Universal Robots PolyScope program: Cobot_soudure_27112023.urp

Program Cobot_soudure_27112023 (installation=Cobot_soudure_27112023 directory=/home/ur/ursim/ursim-5.11.0.108249/programs/TRAVAIL 27112023 createdIn=5.9.4.1031232 lastSavedIn=5.11.0.108249 robotSerialNumber=20195299999)
Calibrated DH parameters: a=[0, -0.6127, -0.57155, 0, 0, 0]; d=[0.1807, 0, 0, 0.17415, 0.11985, 0.11655]; alpha=[1.570796, 0, 0, 1.570796, -1.570796, 0]; deltaTheta=[0, 0, 0, 0, 0, 0]
InitVariablesNode variables(variable(name=Test_Gaz, expression=False), variable(name=Test_Job, expression=False), variable(name=Test_Ordre_Mar, expression=False), variable(name=Valide_Gaz, expression=False), variable(name=fin_soud, expression=1), variable(name=secu_d, expression=0), variable(name=secu_g, expression=0), variable(name=timer_ret_gaz, expression=0))
BeforeStart
  Folder fonctions
    Folder Init [hidden by the author, left out]
    Folder Diverses [hidden by the author, left out]
    Folder Demande [hidden by the author, left out]
    Folder Configuration [hidden by the author, left out]
    Folder Execution [hidden by the author, left out]
    Folder Pas_A_Pas [hidden by the author, left out]
    Folder PopUps
      SuppressedNode
        Folder Configuration [hidden by the author, left out]
      Script file /home/ur/ursim/ursim-5.11.0.108249/programs/SCRIPT/Scripts_soudure/PopUps/Pops_up_PAsAPas.script
        | def pop_up_reg_d():
        |     close_popup()
        |     popup3 = "popup PAS_A_PAS : Table droite programmée"#"popup La table droite est programmée. Appuyer sur le bouton gauche ou droite pour commencer le reglage d'une pièce sur la table associée. La gestion des modes programmation, éxécution et reglage se fait à l'aide des commutateurs superieurs."
        |     socket_open("127.0.0.1",29999,"internal") # open internal socket
        |     socket_send_line(popup3,"internal")     #Affichage message
        |     socket_send_byte(10,"internal")
        | end
        | 
        | def pop_up_reg_g():
        |     close_popup()
        |     popup3 = "popup PAS_A_PAS : Table gauche programmée"#"popup La table gauche est programmée. Appuyer sur le bouton gauche ou droite pour commencer mode pas a pas et le reglage d'une pièce sur la table associée. La gestion des modes programmation, éxécution et reglage se fait à l'aide des commutateurs superieurs."
        |     socket_open("127.0.0.1",29999,"internal") # open internal socket
        |     socket_send_line(popup3,"internal")     #Affichage message
        |     socket_send_byte(10,"internal")
        | end
        | 
        | def pop_up_reg_gd():
        |     close_popup()
        |     popup3 = "popup PAS_A_PAS : Les deux tables sont programmées"#"popup Les deux tables sont programmées. Appuyer sur le bouton gauche ou droite pour commencer le reglage d'une pièce sur la table associée ou passez en mode éxécution à l'aide du commutateur superieur gauche pour effectuer un ou plusieurs cycle(s) de soudure(s)."
        |     socket_open("127.0.0.1",29999,"internal") # open internal socket
        |     socket_send_line(popup3,"internal")     #Affichage message
        |     socket_send_byte(10,"internal")
        | end
        | 
        | def pop_up_reg():
        |     close_popup()
        |     popup3 = "popup PAS_A_PAS : Aucune table n'est programmée"#"popup Appuyer sur le bouton gauche ou droite pour commencer le reglage d'une pièce sur la table associée. La gestion des modes configuration, éxécution et reglage se fait à l'aide des commutateurs superieurs."
        |     socket_open("127.0.0.1",29999,"internal") # open internal socket
        |     socket_send_line(popup3,"internal")     #Affichage message
        |     socket_send_byte(10,"internal")
        | end
        | 
        | def fun_PopUp_PaP(index,type,numPopUP):
        |     index = index +1
        |     char_numeroDeSoudure = to_str(index)
        | 
        |     local resultat = False
        |     local resultat2  = 0
        | 
        |     if (type == 1):
        | 		char_soudure = "point"					#si type = 1, la demande sera sur une soudure point
        | 	elif ((type == 2) or (type ==5)):
        | 		char_soudure = "lineaire"				#si type = 2, la demande sera sur une soudure linéaire
        | 	elif (type == 3):
        | 		char_soudure = "arc de cercle"			#si type = 3, la demande sera sur une soudure arc de cercle
        | 	elif (type == 4):
        | 		char_soudure = "cercle"					#si type = 4, la demande sera sur une soudure cercle
        |     elif (type == 6):
        |         char_soudure = "recopie"                #si type = 5, la demande sera sur une recopie de mouvement
        | 	else :
        | 		char_soudure = "erreur de saisie"
        | 	end
        | 
        |     if (numPopUP == 1):
        |         resultat  = request_boolean_from_primary_client("Soudure numero : " + char_numeroDeSoudure + ", de type : "+ char_soudure + ". Voulez vous effectuer la soudure ?(securité desactivée) Appuyer sur non pour passer à la soudure suivante. ")
        |         return resultat
        |     elif (numPopUP ==2 ):
        |         resultat = request_boolean_from_primary_client("Voulez vous modifier la soudure numéro :" + char_numeroDeSoudure + " ? Appuyez sur non pour continuer")
        |         return resultat
        |     elif (numPopUP ==3 ):
        |         resultat2 = request_integer_from_primary_client("       1-> Point SUIVANT                     Ajouter :    2-> AVANT      3-> APRES")
        |         return resultat2
        |     elif (numPopUP ==4 ):
        |          esultat = request_boolean_from_primary_client("Voulez vous refaire une simulation? Appuyez sur non pour continuer.")
        |         return resultat
        |     end
        | 
        | 
        | end
      Script file /home/ur/ursim/ursim-5.11.0.108249/programs/SCRIPT/Scripts_soudure/PopUps/Pops_up_Execution.script
        | def pop_up_deb_exe_d():
        |     close_popup()
        |     popup3 = "popup Table droite, éxecution... Veillez à bien fermer la porte."
        |     socket_open("127.0.0.1",29999,"internal") # open internal socket
        |     socket_send_line(popup3,"internal")     #Affichage message
        |     socket_send_byte(10,"internal")
        | end
        | 
        | def pop_up_deb_exe_g():
        |     close_popup()
        |     popup3 = "popup Table gauche, éxecution... Veillez à bien fermer la porte."
        |     socket_open("127.0.0.1",29999,"internal") # open internal socket
        |     socket_send_line(popup3,"internal")     #Affichage message
        |     socket_send_byte(10,"internal")
        | end
        | 
        | def pop_up_exe_d():
        |     close_popup()
        |     popup1 = "popup EXECUTION : Table droite prête à éxécution"#"popup Appuyer sur le bouton droit pour commencer l'éxécution de la pièce configurée. La gestion des modes configuration et éxécution se fait à l'aide du commutateur réglage."
        |     socket_open("127.0.0.1",29999,"internal") # open internal socket
        |     socket_send_line(popup1,"internal")     #Affichage message
        |     socket_send_byte(10,"internal")
        | end
        | 
        | def pop_up_exe_g():
        |     close_popup()
        |     popup1 = "popup EXECUTION : Table gauche prête à éxécution"#"popup Appuyer sur le bouton gauche pour commencer l'éxécution de la pièce configurée. La gestion des modes configuration et éxécution se fait à l'aide du commutateur réglage."
        |     socket_open("127.0.0.1",29999,"internal") # open internal socket
        |     socket_send_line(popup1,"internal")     #Affichage message
        |     socket_send_byte(10,"internal")
        | end
        | 
        | def pop_up_fermer_porte():
        |     close_popup()
        |     popup3 = "popup Fermer la porte pour éxecution."
        |     socket_open("127.0.0.1",29999,"internal") # open internal socket
        |     socket_send_line(popup3,"internal")     #Affichage message
        |     socket_send_byte(10,"internal")
        | end
        | 
        | def pop_up_exe():
        |     close_popup()
        |     popup1 ="popup EXECUTION : Les deux tables sont prêtes à l'éxécution" #"popup Appuyer sur le bouton gauche ou droit pour commencer l'éxécution de la pièce sur la table associée. La gestion des modes configuration et éxécution se fait à l'aide du commutateur réglage."
        |     socket_open("127.0.0.1",29999,"internal") # open internal socket
        |     socket_send_line(popup1,"internal")     #Affichage message
        |     socket_send_byte(10,"internal")
        | end
      Script file /home/ur/ursim/ursim-5.11.0.108249/programs/SCRIPT/Scripts_soudure/PopUps/Pops_up_Configuration.script
        | def pop_up_config():
        |     close_popup()
        |     popup3 = "popup CONFIGURATION : Aucune table de configurée."
        |     socket_open("127.0.0.1",29999,"internal") # open internal socket
        |     socket_send_line(popup3,"internal")     #Affichage message
        |     socket_send_byte(10,"internal")
        | end
        | 
        | def pop_up_config_d():
        |     close_popup()
        |     popup3 = "popup CONFIGURATION : Table droite configurée."
        |     socket_open("127.0.0.1",29999,"internal") # open internal socket
        |     socket_send_line(popup3,"internal")     #Affichage message
        |     socket_send_byte(10,"internal")
        | end
        | 
        | def pop_up_config_g_et_d():
        |     close_popup()
        |     popup3 = "popup CONFIGURATION : Les deux tables sont configurées."
        |     socket_open("127.0.0.1",29999,"internal") # open internal socket
        |     socket_send_line(popup3,"internal")     #Affichage message
        |     socket_send_byte(10,"internal")
        | end
        | 
        | def pop_up_config_g():
        |     close_popup()
        |     popup3 = "popup CONFIGURATION : Table droite configurée."
        |     socket_open("127.0.0.1",29999,"internal") # open internal socket
        |     socket_send_line(popup3,"internal")     #Affichage message
        |     socket_send_byte(10,"internal")
        | end
      SuppressedNode
        Folder Execution [hidden by the author, left out]
      SuppressedNode
        Folder Pas_A_Pas [hidden by the author, left out]
    Folder Mouvements soudures [hidden by the author, left out]
Robot Program (runOnlyOnce=true)
  SuppressedNode
    Folder Initialisation
      Loop Counting (count=1) loopVariable(name=Boucle_10)
        Script: fun_adresse_bp()
  Script file /home/ur/ursim/ursim-5.11.0.108249/programs/SCRIPT/Scripts_soudure/general.script
    | while (True):
    |   # 68 "Programme de robot"
    |   global safe_mode=0
    | 
    |   set_configurable_digital_out(0, False)
    | 
    |   set_configurable_digital_out(1, False)
    | 
    |   while (get_configurable_digital_in(4) ==   True    or  get_configurable_digital_in(5) ==   True  ):
    | 
    |     sync()
    |     # 94 "'clingottement pour signifier qu'il y  un defaut sur un des carters '"
    |     set_standard_digital_out(4, False)
    |     set_configurable_digital_out(6, False)
    |     sleep(0.5)
    |     set_standard_digital_out(4, True)
    |     set_configurable_digital_out(6, True)
    |     sleep(0.5)
    |     sync()
    |   end
    | 
    |   set_configurable_digital_out(6, False)
    |   set_standard_digital_out(4, False)
    |   sleep(2.0)
    |   #movel(pose_add(get_target_tcp_pose(), pose_sub(PointPassage_12_to_p, PointPassage_12_from_p)), a=0.01, v=2.0E-4)
    |   global angle_base= get_actual_joint_positions ()
    |   if (angle_base[0]  <= 0.7):
    |     if (angle_base[0] >= 1.6):
    |       # 116 "Départ"        A CHANGER PAR UNE POSTION ENREGISTREE
    |       movej([0.7376820445060732, 1.3357652919721463, -2.8533326461405863, -0.44459326684985356, 1.9245067834854124, 4.003490924835204], a=1.3962634015954636, v=1.0471975511965976)
    |     else:
    |       if (angle_base[0]>1.6):
    |         movej(Point_init_D, a=1.3962634015954636, v=1.7453292519943295)
    |         movej(Point_avt_initD, a=1.3962634015954636, v=1.7453292519943295)
    |       else:
    |         if (angle_base[0]<0.7):
    |           movej(Point_init_G, a=1.3962634015954636, v=1.7453292519943295)
    |         end
    |       end
    |     end
    |   else:
    |     # 124 "SinonSi angle_base[0]>1.6"
    |     if (angle_base[0]>1.6):
    | 
    |       movej(Point_init_D, a=1.3962634015954636, v=1.7453292519943295)
    |       movej(Point_avt_initD, a=1.3962634015954636, v=1.7453292519943295)
    |     else:
    |       if (angle_base[0]<0.7):
    |         movej(Point_init_G, a=1.3962634015954636, v=1.7453292519943295)
    |       end
    |     end
    |   end
    |   # 131 "Départ"             A CHANGER PAR UNE POSTION ENREGISTREE
    |   movej([0.7376820445060732, 1.3357652919721463, -2.8533326461405863, -0.44459326684985356, 1.9245067834854124, 4.003490924835204], a=1.3962634015954636, v=1.0471975511965976)
    |   global angle_base= get_actual_joint_positions ()
    |   # 'mode config'
    |   if (get_configurable_digital_in(7)  ==   False    and  get_standard_digital_in(7)  ==   False  ):
    |     if ((config_g  ==  1)   and   (config_d  ==  1)):
    |       pop_up_config_g_et_d()
    |     else:
    |       if ((config_g  == 1)):
    |         pop_up_config_g()
    |       else:
    |         if (config_d  ==  1):
    |           pop_up_config_d()
    |         else:
    |           if ((config_g  ==  0)  and  (config_d  ==  0)):
    |             pop_up_config()
    |           end
    |         end
    |       end
    |     end
    |     global boucle=1
    |     while ((get_configurable_digital_in(7)  ==   False  )  and  (boucle  ==  1)   and  (get_standard_digital_in(7) ==   False  )):
    |       thread Thread_while_145():
    |         while (True):
    |           set_standard_digital_out(5, True)
    |           set_standard_digital_out(6, False)
    |           sleep(0.5)
    |           set_standard_digital_out(5, False)
    |           set_standard_digital_out(6, True)
    |           sleep(0.5)
    |           sync()
    |         end
    |       end
    |       if (get_standard_digital_in(3) ==   False    and  get_standard_digital_in(2) ==   False    and  get_configurable_digital_in(7)  ==    False    and  get_standard_digital_in(7) ==   False  ):
    |         global thread_handler_145=run Thread_while_145()
    |         while (get_standard_digital_in(3) ==   False    and  get_standard_digital_in(2) ==   False    and  get_configurable_digital_in(7)  ==    False    and  get_standard_digital_in(7) ==   False  ):
    |           sync()
    |         end
    |         kill thread_handler_145
    |       end
    |       if (get_standard_digital_in(2)  ==   True  ):
    |         set_standard_digital_out(5, True)
    |         set_standard_digital_out(6, False)
    |         movej(Point_init_G, a=1.3962634015954636, v=1.0471975511965976, r=0.006)
    |         movej(Point_Attente_G, a=1.3962634015954636, v=1.0471975511965976, r=0.006)
    |         movej(Point_config_g, a=0.6981317007977318, v=0.5235987755982988)
    |         global led_cobot=1
    |         fun_config_g()
    |         global led_cobot=0
    |         fun_valid_config_g()
    |         movej(Point_Attente_G, a=1.3962634015954636, v=1.0471975511965976, r=0.006)
    |         movej(Point_init_G, a=1.3962634015954636, v=1.0471975511965976, r=0.006)
    |         # 170 "Départ"         A CHANGER PAR UNE POSTION ENREGISTREE
    |         movej([0.7376820445060732, 1.3357652919721463, -2.8533326461405863, -0.44459326684985356, 1.9245067834854124, 4.003490924835204], a=1.3962634015954636, v=1.0471975511965976)
    |       end
    | 
    |       if (get_standard_digital_in(3)  ==   True  ):
    |         set_standard_digital_out(6, True)
    |         set_standard_digital_out(5, False)
    |         movej(Point_avt_initD, a=1.3962634015954636, v=1.0471975511965976, r=0.006)
    |         movej(Point_init_D, a=1.3962634015954636, v=1.0471975511965976)
    |         movej(Point_Attente_D, a=1.3962634015954636, v=1.0471975511965976, r=0.006)
    |         movej(Point_config_d, a=0.6981317007977318, v=0.5235987755982988)
    |         global led_cobot=1
    |         fun_config_d()
    |         global led_cobot=0
    |         fun_valid_config_d()
    |         movej(Point_Attente_D, a=1.3962634015954636, v=1.0471975511965976, r=0.006)
    |         movej(Point_init_D, a=1.3962634015954636, v=1.0471975511965976, r=0.006)
    |         movej(Point_avt_initD, a=1.3962634015954636, v=1.0471975511965976, r=0.006)
    |         # 190 "Départ"         A CHANGER PAR UNE POSTION ENREGISTREE
    |         movej([0.7376820445060732, 1.3357652919721463, -2.8533326461405863, -0.44459326684985356, 1.9245067834854124, 4.003490924835204], a=1.3962634015954636, v=1.0471975511965976)
    |       end
    |     end
    |   end
    |   # '"Reglage"'
    | 
    |   if (get_configurable_digital_in(7)  ==   False    and  get_standard_digital_in(7)  ==   True  ):
    |     if ((config_g  ==  1)   and   (config_d  ==  1)):
    |       pop_up_reg_gd()
    |       global boucle=1
    |     else:
    |       if (config_g  ==  1):
    |         pop_up_reg_gd()
    |         global boucle=1
    |       else:
    |         if (config_d  ==  1):
    |           pop_up_reg_d()
    |           global boucle=1
    |         else:
    |           close_popup()
    |           while (get_standard_digital_in(7)  ==   True  ):
    |             popup("Aucune configuration n'est actuellement detectée.", "Erreur", False, True, blocking=True)
    |           end
    |         end
    |       end
    |     end
    |     global boucle=1
    |     while ((get_configurable_digital_in(7)  ==   False  )  and  (boucle  ==  1)   and  (get_standard_digital_in(7) ==   True  )):
    |       thread Thread_while_208():
    |         while (True):
    |           if (config_g  ==  1):
    |             set_standard_digital_out(5, True)
    |           end
    |           if (config_d  ==  1):
    |             set_standard_digital_out(6, True)
    |           end
    |           sleep(0.5)
    |           set_standard_digital_out(5, False)
    |           set_standard_digital_out(6, False)
    |           sleep(0.5)
    |         end
    |       end
    |       if (get_standard_digital_in(3) ==   False    and  get_standard_digital_in(2) ==   False    and  get_configurable_digital_in(7)  ==    False    and  get_standard_digital_in(7)  ==   True  ):
    |         global thread_handler_208=run Thread_while_208()
    |         while (get_standard_digital_in(3) ==   False    and  get_standard_digital_in(2) ==   False    and  get_configurable_digital_in(7)  ==    False    and  get_standard_digital_in(7)  ==   True  ):
    |           sync()
    |         end
    |         kill thread_handler_208
    |       end
    |       if (get_standard_digital_in(2)  ==   True  ):
    |         global safe_mode=1
    |         set_standard_digital_out(5, True)
    |         set_standard_digital_out(6, False)
    |         movej(Point_init_G, a=1.3962634015954636, v=1.0471975511965976, r=0.006)
    |         movej(Point_Attente_G, a=1.3962634015954636, v=1.0471975511965976, r=0.006)
    |         movej(pose_inter_g, a=0.6981317007977318, v=0.5235987755982988)
    |         global led_cobot=1
    |         fun_Pas_A_Pas_g()
    |         global led_cobot=0
    |         global safe_mode=0
    |         global boucle=0
    |       end
    |       if (get_standard_digital_in(3)  ==   True  ):
    |         global safe_mode=1
    |         set_standard_digital_out(6, True)
    |         set_standard_digital_out(5, False)
    |         movej(Point_avt_initD, a=1.3962634015954636, v=1.0471975511965976, r=0.006)
    |         movej(Point_init_D, a=1.3962634015954636, v=1.0471975511965976, r=0.006)
    |         movej(pose_inter_d, a=0.6981317007977318, v=0.5235987755982988)
    |         global led_cobot=1
    |         fun_Pas_A_Pas_d()
    |         global led_cobot=0
    |         global safe_mode=0
    |         global boucle=0
    |       end
    |     end
    |   end
    |   # 'mode execution'
    |   if (get_configurable_digital_in(7)  ==   True  ):
    |     if ((config_g  ==  1)   and   (config_d  ==  1)):
    |       pop_up_exe()
    |       global boucle=1
    |     else:
    |       if (config_g  ==  1):
    |         pop_up_exe_g()
    |         global boucle=1
    |       else:
    |         if (config_d  ==  1):
    |           pop_up_exe_d()
    |           global boucle=1
    |         else:
    |           close_popup()
    |           while (get_configurable_digital_in(7)  ==   True  ):
    |             popup("Aucune programmation n'est actuellement detectée, veillez à programmer une pièce avant de vouloir l'éxécuter.", "Erreur", False, True, blocking=True)
    |           end
    |         end
    |       end
    |     end
    |     while (( get_configurable_digital_in(7)  ==   True  )   and  (boucle  ==  1)):
    |       thread Thread_while_259():
    |         while (True):
    |           if (config_g  ==  1):
    |             set_standard_digital_out(5, True)
    |           end
    |           if (config_d  ==  1):
    |             set_standard_digital_out(6, True)
    |           end
    |           sleep(0.5)
    |           set_standard_digital_out(5, False)
    |           set_standard_digital_out(6, False)
    |           sleep(0.5)
    |         end
    |       end
    |       if (get_standard_digital_in(3) ==   False    and  get_standard_digital_in(2) ==   False    and  get_configurable_digital_in(7) ==   True  ):
    |         global thread_handler_259=run Thread_while_259()
    |         while (get_standard_digital_in(3) ==   False    and  get_standard_digital_in(2) ==   False    and  get_configurable_digital_in(7) ==   True  ):
    |           sync()
    |         end
    |         kill thread_handler_259
    |       end
    |       if ((get_standard_digital_in(2)  ==   True  )  and  (config_g  ==   True  )):
    |         global boucle_g=1
    |         while (boucle_g  ==  1):
    |           set_configurable_digital_out(0, True)
    |           set_standard_digital_out(5, True)
    |           set_standard_digital_out(6, False)
    |           sleep(0.25)
    |           set_standard_digital_out(5, False)
    |           sleep(0.25)
    |           if (get_configurable_digital_in(4)  ==    False  ):
    |             set_standard_digital_out(5, True)
    |             if (get_configurable_digital_in(4)  ==    False  ):
    |               close_popup()
    |               while (get_configurable_digital_in(4) == False):
    |                 sync()
    |               end
    |             end
    |           end
    |           if (get_configurable_digital_in(4)  ==    True  ):
    |             global secu_g=1
    |             set_standard_digital_out(5, True)
    |             movej(Point_init_G, a=1.3962634015954636, v=1.0471975511965976, r=0.006)
    |             fun_execution_g()
    |             movej(Point_Attente_G, a=1.3962634015954636, v=1.0471975511965976, r=0.006)
    |             movej(Point_init_G, a=1.3962634015954636, v=1.0471975511965976, r=0.006)
    |             # 294 "Départ"         A CHANGER PAR UNE POSTION ENREGISTREE
    |             movej([0.7376820445060732, 1.3357652919721463, -2.8533326461405863, -0.44459326684985356, 1.9245067834854124, 4.003490924835204], a=1.3962634015954636, v=1.0471975511965976)
    |             set_configurable_digital_out(0, False)
    |             global secu_g=0
    |             global boucle_g=0
    |           end
    |         end
    |         global boucle=0
    |       else:
    |         if ((get_standard_digital_in(2)  ==   True  )  and  (config_g  ==   False  )):
    |           close_popup()
    |           popup("Aucune programmation n'est actuellement detectée sur la table gauche, veillez à programmer une pièce avant de vouloir l'éxécuter.", "Erreur", False, True, blocking=True)
    |           global boucle=0
    |         end
    |       end
    |       if ((get_standard_digital_in(3)  ==   True  )  and  (config_d  ==   True  )):
    |         global boucle_d=1
    |         pop_up_deb_exe_d()
    |         while (boucle_d  ==  1):
    |           set_configurable_digital_out(1, True)
    |           set_standard_digital_out(5, False)
    |           set_standard_digital_out(6, True)
    |           sleep(0.25)
    |           set_standard_digital_out(6, False)
    |           sleep(0.25)
    |           if (get_configurable_digital_in(5)  ==    False  ):
    |             set_standard_digital_out(6, True)
    |             sleep(6.0)
    |             if (get_configurable_digital_in(5)  ==    False  ):
    |               close_popup()
    |               while (get_configurable_digital_in(5) == False):
    |                 sync()
    |               end
    |             end
    |           end
    |           if (get_configurable_digital_in(5)  ==    True  ):
    |             global secu_d=1
    |             set_standard_digital_out(6, True)
    |             movej(Point_avt_initD, a=1.3962634015954636, v=1.0471975511965976)
    |             fun_execution_d()
    |             set_configurable_digital_out(1, False)
    |             global secu_d=0
    |             global boucle_d=0
    |           end
    |         end
    |         global boucle=0
    |       else:
    |         if ((get_standard_digital_in(3)  ==   True  )  and  (config_d  ==   False  )):
    |           close_popup()
    |           popup("Aucune programmation n'est actuellement detectée sur la table droite, veillez à programmer une pièce avant de vouloir l'éxécuter.", "Erreur", False, True, blocking=True)
    |           global boucle=0
    |         end
    |       end
    |     end
    |   end
    | end
    | end
  SuppressedNode
    MoveJ speed 60 deg/s, acceleration 80 deg/s^2 (useActiveTCP=true) feature=Base
      SafeHome (positionOptionType=SPEED_AND_ACCELERATION speed=1.047198 acceleration=1.396263 nextMotionTime=2)
      Waypoint Waypoint (Variable): motionParameters(jointSpeed=0.523599 jointAcceleration=0.698132 cartesianSpeed=0.25 cartesianAcceleration=1.2); variable(featureName=Point_init_G)
      Waypoint Waypoint (Variable): motionParameters(jointSpeed=0.523599 jointAcceleration=0.698132 cartesianSpeed=0.25 cartesianAcceleration=1.2); variable(featureName=Point_Attente_G)
      Waypoint Waypoint (Variable): motionParameters(jointSpeed=0.523599 jointAcceleration=0.698132 cartesianSpeed=0.25 cartesianAcceleration=1.2); variable(featureName=Point_config_g)
      Waypoint Waypoint (Variable): motionParameters(jointSpeed=0.523599 jointAcceleration=0.698132 cartesianSpeed=0.25 cartesianAcceleration=1.2); variable(featureName=Point_Attente_G)
      Waypoint Waypoint (Variable): motionParameters(jointSpeed=0.523599 jointAcceleration=0.698132 cartesianSpeed=0.25 cartesianAcceleration=1.2); variable(featureName=Point_init_G)
      SafeHome (positionOptionType=SPEED_AND_ACCELERATION speed=1.047198 acceleration=1.396263 nextMotionTime=2)
      Waypoint Waypoint (Variable): motionParameters(jointSpeed=0.785398 jointAcceleration=1.047198 cartesianSpeed=0.25 cartesianAcceleration=1.2); variable(featureName=Point_avt_initD)
      Waypoint Waypoint (Variable): motionParameters(jointSpeed=0.523599 jointAcceleration=0.698132 cartesianSpeed=0.25 cartesianAcceleration=1.2); variable(featureName=Point_init_D)
      Waypoint Waypoint (Variable): motionParameters(jointSpeed=0.523599 jointAcceleration=0.698132 cartesianSpeed=0.25 cartesianAcceleration=1.2); variable(featureName=Point_Attente_D)
      Waypoint Waypoint (Variable): motionParameters(jointSpeed=0.523599 jointAcceleration=0.698132 cartesianSpeed=0.25 cartesianAcceleration=1.2); variable(featureName=Point_config_d)
      Waypoint Waypoint (Variable): motionParameters(jointSpeed=0.523599 jointAcceleration=0.698132 cartesianSpeed=0.25 cartesianAcceleration=1.2); variable(featureName=Point_Attente_D)
      Waypoint Waypoint (Variable): motionParameters(jointSpeed=0.523599 jointAcceleration=0.698132 cartesianSpeed=0.25 cartesianAcceleration=1.2); variable(featureName=Point_init_D)
      SafeHome (positionOptionType=SPEED_AND_ACCELERATION speed=1.047198 acceleration=1.396263 nextMotionTime=2)
  SuppressedNode
    safe_mode := 0
  SuppressedNode
    Folder Deplacement vers position initial
      SuppressedNode
        Popup Message (haltProgram=false message=debut deplacement vers position initiale inputType=Text)
      Set DigitalOutput pin=Cmd_Carter_Bit1; digitalValue=0
      Set DigitalOutput pin=Cmd_Carter_Bit2; digitalValue=0
      Loop While (checkContinuously=false) expression=SecuGaucheOk≟ True  or SecuDroiteOk≟ True
        Script: sync()
        'clingottement pour signifier qu'il y  un defaut sur un des carters '
        Set DigitalOutput pin=Dcy_Voyant; digitalValue=0
        Set DigitalOutput pin=Led_Arret; digitalValue=0
        Wait Sleep waitTime=0.5
        Set DigitalOutput pin=Dcy_Voyant; digitalValue=1
        Set DigitalOutput pin=Led_Arret; digitalValue=1
        Wait Sleep waitTime=0.5
      Set DigitalOutput pin=Led_Arret; digitalValue=0
      Set DigitalOutput pin=Dcy_Voyant; digitalValue=0
      Wait Sleep waitTime=2
      'etre sur de l'ouverture complete du carter '
      MoveL speed 0.2 mm/s, acceleration 10 mm/s^2 (useActiveTCP=true) feature=Base
        Waypoint PointPassage_12 (Relative): relativeFromPosition TCP in base x=100.468 y=319.613 z=576.47 mm, rx=-0.0214 ry=-0.0122 rz=1.5415 rad; joints [-139.419, 75.739, -163.156, -3.26, 89.083, -42.172] deg; TCP offset x=-8.331 y=2.512 z=301.573 mm, rx=0 ry=0 rz=0 rad; TCP in base x=100.463 y=319.639 z=576.462 mm, rx=-0.0214 ry=-0.0122 rz=1.5416 rad; joints [-139.419, 75.741, -163.155, -3.263, 89.08, -42.17] deg
        'Pos_cobot a etait affectuer a la position init (l3)'
        'Pos_cobot[2] correspond a la valeur Z de la postion init (l4)'
      SuppressedNode
        MoveJ speed 60 deg/s, acceleration 80 deg/s^2 (useActiveTCP=true) feature=Base
          SuppressedNode
            Waypoint Position_init: motionParameters(jointSpeed=1.047198 jointAcceleration=1.396263 cartesianSpeed=0.25 cartesianAcceleration=1.2); TCP in base x=96.613 y=317.698 z=575.432 mm, rx=-0.0254 ry=-0.0254 rz=1.5393 rad; joints [-139.566, 75.575, -163.284, -3.665, 88.92, -42.143] deg; TCP offset x=-6.782 y=1.742 z=298.685 mm, rx=0 ry=0 rz=0 rad
          SuppressedNode
            Waypoint Waypoint (Variable): variable(featureName=Point_init)
          'Apres avoir eu la position du robot et tester la valeur de Z pour faire un mouvement verticale on envoi le robot en position init'
      angle_base := get_actual_joint_positions()
      If angle_base[0] ≤0.7
        If angle_base[0]≥1.6
          SafeHome (positionOptionType=SPEED_AND_ACCELERATION speed=1.047198 acceleration=1.396263 nextMotionTime=2)
        ElseIf angle_base[0]>1.6
          MoveJ speed 100 deg/s, acceleration 80 deg/s^2 (useActiveTCP=true) feature=Base
            Waypoint Waypoint (Variable): variable(featureName=Point_init_D)
            Waypoint Waypoint (Variable): variable(featureName=Point_avt_initD)
        ElseIf angle_base[0]<0.7
          MoveJ speed 100 deg/s, acceleration 80 deg/s^2 (useActiveTCP=true) feature=Base
            Waypoint Waypoint (Variable): variable(featureName=Point_init_G)
      ElseIf angle_base[0]>1.6
        MoveJ speed 100 deg/s, acceleration 80 deg/s^2 (useActiveTCP=true) feature=Base
          Waypoint Waypoint (Variable): variable(featureName=Point_init_D)
          Waypoint Waypoint (Variable): variable(featureName=Point_avt_initD)
      ElseIf angle_base[0]<0.7
        MoveJ speed 100 deg/s, acceleration 80 deg/s^2 (useActiveTCP=true) feature=Base
          Waypoint Waypoint (Variable): variable(featureName=Point_init_G)
      SafeHome (positionOptionType=SPEED_AND_ACCELERATION speed=1.047198 acceleration=1.396263 nextMotionTime=2)
      angle_base := get_actual_joint_positions()
  SuppressedNode
    'mode config'
  SuppressedNode
    If Mode_manu ≟ False  and config_reglage ≟ False
      If (config_g ≟ 1)  and  (config_d ≟ 1)
        Script: pop_up_config_g_et_d()
      ElseIf (config_g ≟1)
        Script: pop_up_config_g()
      ElseIf config_d ≟ 1
        Script: pop_up_config_d()
      ElseIf (config_g ≟ 0) and (config_d ≟ 0)
        Script: pop_up_config()
      boucle := 1
      Loop While (checkContinuously=false) expression=(Mode_manu ≟ False ) and (boucle ≟ 1)  and (config_reglage≟ False )
        Loop While (checkContinuously=true) expression=Pret_Table_Droi≟ False  and Pret_Table_Gauc≟ False  and Mode_manu ≟  False  and config_reglage≟ False
          Set DigitalOutput pin=Voyant_Table_Ga; digitalValue=1
          Set DigitalOutput pin=Voyant_Table_Dr; digitalValue=0
          Wait Sleep waitTime=0.5
          Set DigitalOutput pin=Voyant_Table_Ga; digitalValue=0
          Set DigitalOutput pin=Voyant_Table_Dr; digitalValue=1
          Wait Sleep waitTime=0.5
          Script: sync()
        If Pret_Table_Gauc ≟ True
          Set DigitalOutput pin=Voyant_Table_Ga; digitalValue=1
          Set DigitalOutput pin=Voyant_Table_Dr; digitalValue=0
          'plus de demande du nombre de point a saisir'
          MoveJ speed 60 deg/s, acceleration 80 deg/s^2 (useActiveTCP=true) feature=Base
            Waypoint Waypoint (Variable): motionParameters(blendRadius=0.006); variable(featureName=Point_init_G)
            Waypoint Waypoint (Variable): motionParameters(blendRadius=0.006); variable(featureName=Point_Attente_G)
            Waypoint Waypoint (Variable): motionParameters(jointSpeed=0.523599 jointAcceleration=0.698132 cartesianSpeed=0.25 cartesianAcceleration=1.2); variable(featureName=Point_config_g)
            led_cobot := 1
            Script: fun_config_g()
            led_cobot := 0
            Script: fun_valid_config_g()
            MoveJ speed 60 deg/s, acceleration 80 deg/s^2 (useActiveTCP=true) feature=Base
              SuppressedNode
                Waypoint anti_poq_g: motionParameters(jointSpeed=0.523599 jointAcceleration=0.698132 cartesianSpeed=0.25 cartesianAcceleration=1.2 blendRadius=0.07); TCP in base x=433.126 y=153.22 z=577.202 mm, rx=0.0572 ry=-0.0147 rz=1.5652 rad; joints [-179.123, 70.738, -150.145, -9.057, 92.825, -1.059] deg; TCP offset x=-8.331 y=2.512 z=301.573 mm, rx=0 ry=0 rz=0 rad
              Waypoint Waypoint (Variable): motionParameters(blendRadius=0.006); variable(featureName=Point_Attente_G)
              Waypoint Waypoint (Variable): motionParameters(blendRadius=0.006); variable(featureName=Point_init_G)
              SuppressedNode
                Waypoint Waypoint (Variable): motionParameters(jointSpeed=0.523599 jointAcceleration=0.698132 cartesianSpeed=0.25 cartesianAcceleration=1.2); variable(featureName=Point_init)
              SafeHome (positionOptionType=SPEED_AND_ACCELERATION speed=1.047198 acceleration=1.396263 nextMotionTime=2)
        If Pret_Table_Droi ≟ True
          Set DigitalOutput pin=Voyant_Table_Dr; digitalValue=1
          Set DigitalOutput pin=Voyant_Table_Ga; digitalValue=0
          MoveJ speed 60 deg/s, acceleration 80 deg/s^2 (useActiveTCP=true) feature=Base
            Waypoint Waypoint (Variable): motionParameters(blendRadius=0.006); variable(featureName=Point_avt_initD)
            Waypoint Waypoint (Variable): variable(featureName=Point_init_D)
            Waypoint Waypoint (Variable): motionParameters(blendRadius=0.006); variable(featureName=Point_Attente_D)
            Waypoint Waypoint (Variable): motionParameters(jointSpeed=0.523599 jointAcceleration=0.698132 cartesianSpeed=0.25 cartesianAcceleration=1.2); variable(featureName=Point_config_d)
          led_cobot := 1
          Script: fun_config_d()
          led_cobot := 0
          Script: fun_valid_config_d()
          MoveJ speed 60 deg/s, acceleration 80 deg/s^2 (useActiveTCP=true) feature=Base
            SuppressedNode
              Waypoint anti_poq_1_d: motionParameters(jointSpeed=0.523599 jointAcceleration=0.698132 cartesianSpeed=0.25 cartesianAcceleration=1.2 blendRadius=0); TCP in base x=-432.081 y=47.828 z=581.386 mm, rx=0.0024 ry=-0.0004 rz=1.5709 rad; joints [-31.202, 71.743, -153.151, -8.683, 90.121, -148.72] deg
            SuppressedNode
              Waypoint anti_poq_2_d: motionParameters(jointSpeed=1.047198 jointAcceleration=1.396263 cartesianSpeed=0.25 cartesianAcceleration=1.2 blendRadius=0.07); TCP in base x=-292.604 y=310.313 z=583.956 mm, rx=-0.0324 ry=-0.0877 rz=3.0963 rad; joints [-72.124, 71.739, -151.869, -12.519, 87.987, -20.279] deg; TCP offset x=-8.331 y=2.512 z=301.573 mm, rx=0 ry=0 rz=0 rad
            SuppressedNode
              Waypoint Waypoint (Variable): motionParameters(jointSpeed=0.785398 jointAcceleration=1.047198 cartesianSpeed=0.25 cartesianAcceleration=1.2); variable(featureName=Point_init)
            Waypoint Waypoint (Variable): motionParameters(blendRadius=0.006); variable(featureName=Point_Attente_D)
            Waypoint Waypoint (Variable): motionParameters(blendRadius=0.006); variable(featureName=Point_init_D)
            Waypoint Waypoint (Variable): motionParameters(blendRadius=0.006); variable(featureName=Point_avt_initD)
            SafeHome (positionOptionType=SPEED_AND_ACCELERATION speed=1.047198 acceleration=1.396263 nextMotionTime=2)
  SuppressedNode
    '"Reg"'
  SuppressedNode
    If Mode_manu ≟ False  and config_reglage ≟ True
      If (config_g ≟ 1)  and  (config_d ≟ 1)
        Script: pop_up_reg_gd()
        boucle := 1
      ElseIf config_g ≟ 1
        Script: pop_up_reg_gd()
        boucle := 1
      ElseIf config_d ≟ 1
        Script: pop_up_reg_d()
        boucle := 1
      Else 
        Script: close_popup()
        Loop While (checkContinuously=false) expression=config_reglage ≟ True
          Popup Error (haltProgram=false message=Aucune configuration n'est actuellement detectée. inputType=Text)
      boucle := 1
      Loop While (checkContinuously=false) expression=(Mode_manu ≟ False ) and (boucle ≟ 1)  and (config_reglage≟ True )
        Loop While (checkContinuously=true) expression=Pret_Table_Droi≟ False  and Pret_Table_Gauc≟ False  and Mode_manu ≟  False  and config_reglage ≟ True
          If config_g ≟ 1
            Set DigitalOutput pin=Voyant_Table_Ga; digitalValue=1
          If config_d ≟ 1
            Set DigitalOutput pin=Voyant_Table_Dr; digitalValue=1
          Wait Sleep waitTime=0.5
          Set DigitalOutput pin=Voyant_Table_Ga; digitalValue=0
          Set DigitalOutput pin=Voyant_Table_Dr; digitalValue=0
          Wait Sleep waitTime=0.5
        If Pret_Table_Gauc ≟ True
          safe_mode := 1
          Set DigitalOutput pin=Voyant_Table_Ga; digitalValue=1
          Set DigitalOutput pin=Voyant_Table_Dr; digitalValue=0
          MoveJ speed 60 deg/s, acceleration 80 deg/s^2 (useActiveTCP=true) feature=Base
            Waypoint Waypoint (Variable): motionParameters(blendRadius=0.006); variable(featureName=Point_init_G)
            Waypoint Waypoint (Variable): motionParameters(blendRadius=0.006); variable(featureName=Point_Attente_G)
            Waypoint Waypoint (Variable): motionParameters(jointSpeed=0.523599 jointAcceleration=0.698132 cartesianSpeed=0.25 cartesianAcceleration=1.2); variable(featureName=pose_inter_g)
          led_cobot := 1
          Script: fun_Pas_A_Pas_g()
          led_cobot := 0
          safe_mode := 0
          boucle := 0
        If Pret_Table_Droi ≟ True
          safe_mode := 1
          Set DigitalOutput pin=Voyant_Table_Dr; digitalValue=1
          Set DigitalOutput pin=Voyant_Table_Ga; digitalValue=0
          MoveJ speed 60 deg/s, acceleration 80 deg/s^2 (useActiveTCP=true) feature=Base
            Waypoint Waypoint (Variable): motionParameters(blendRadius=0.006); variable(featureName=Point_avt_initD)
            Waypoint Waypoint (Variable): motionParameters(blendRadius=0.006); variable(featureName=Point_init_D)
            Waypoint Waypoint (Variable): motionParameters(jointSpeed=0.523599 jointAcceleration=0.698132 cartesianSpeed=0.25 cartesianAcceleration=1.2); variable(featureName=pose_inter_d)
          led_cobot := 1
          Script: fun_Pas_A_Pas_d()
          led_cobot := 0
          safe_mode := 0
          boucle := 0
  SuppressedNode
    'mode exe'
  SuppressedNode
    If Mode_manu ≟ True
      If (config_g ≟ 1)  and  (config_d ≟ 1)
        Script: pop_up_exe()
        boucle := 1
      ElseIf config_g ≟ 1
        Script: pop_up_exe_g()
        boucle := 1
      ElseIf config_d ≟ 1
        Script: pop_up_exe_d()
        boucle := 1
      Else 
        Script: close_popup()
        Loop While (checkContinuously=false) expression=Mode_manu ≟ True
          Popup Error (haltProgram=false message=Aucune programmation n'est actuellement detectée, veillez à programmer une pièce avant de vouloir l'éxécuter. inputType=Text)
      Loop While (checkContinuously=false) expression=( Mode_manu ≟ True )  and (boucle ≟ 1)
        Loop While (checkContinuously=true) expression=Pret_Table_Droi≟ False  and Pret_Table_Gauc≟ False  and Mode_manu≟ True
          If config_g ≟ 1
            Set DigitalOutput pin=Voyant_Table_Ga; digitalValue=1
          If config_d ≟ 1
            Set DigitalOutput pin=Voyant_Table_Dr; digitalValue=1
          Wait Sleep waitTime=0.5
          Set DigitalOutput pin=Voyant_Table_Ga; digitalValue=0
          Set DigitalOutput pin=Voyant_Table_Dr; digitalValue=0
          Wait Sleep waitTime=0.5
        If (Pret_Table_Gauc ≟ True ) and (config_g ≟ True )
          boucle_g := 1
          SuppressedNode
            Script: pop_up_deb_exe_g()
          Loop While (checkContinuously=false) expression=boucle_g ≟ 1
            Set DigitalOutput pin=Cmd_Carter_Bit1; digitalValue=1
            Set DigitalOutput pin=Voyant_Table_Ga; digitalValue=1
            Set DigitalOutput pin=Voyant_Table_Dr; digitalValue=0
            Wait Sleep waitTime=0.25
            Set DigitalOutput pin=Voyant_Table_Ga; digitalValue=0
            Wait Sleep waitTime=0.25
            If SecuGaucheOk ≟  False
              Set DigitalOutput pin=Voyant_Table_Ga; digitalValue=1
              SuppressedNode
                Wait Sleep waitTime=6
              If SecuGaucheOk ≟  False
                Script: close_popup()
                Wait DigitalInput pin=SecuGaucheOk; digitalValue=1
            If SecuGaucheOk ≟  True
              secu_g := 1
              Set DigitalOutput pin=Voyant_Table_Ga; digitalValue=1
              MoveJ speed 60 deg/s, acceleration 80 deg/s^2 (useActiveTCP=true) feature=Base
                Waypoint Waypoint (Variable): motionParameters(blendRadius=0.006); variable(featureName=Point_init_G)
                SuppressedNode
                  Waypoint Waypoint (Variable): motionParameters(blendRadius=0.006); variable(featureName=Point_Attente_G)
              Script: fun_execution_g()
              MoveJ speed 60 deg/s, acceleration 80 deg/s^2 (useActiveTCP=true) feature=Base
                Waypoint Waypoint (Variable): motionParameters(blendRadius=0.006); variable(featureName=Point_Attente_G)
                Waypoint Waypoint (Variable): motionParameters(blendRadius=0.006); variable(featureName=Point_init_G)
                SafeHome (positionOptionType=SPEED_AND_ACCELERATION speed=1.047198 acceleration=1.396263 nextMotionTime=2)
              Set DigitalOutput pin=Cmd_Carter_Bit1; digitalValue=0
              secu_g := 0
              boucle_g := 0
          boucle := 0
        ElseIf (Pret_Table_Gauc ≟ True ) and (config_g ≟ False )
          Script: close_popup()
          Popup Error (haltProgram=false message=Aucune programmation n'est actuellement detectée sur la table gauche, veillez à programmer une pièce avant de vouloir l'éxécuter. inputType=Text)
          boucle := 0
        If (Pret_Table_Droi ≟ True ) and (config_d ≟ True )
          boucle_d := 1
          Script: pop_up_deb_exe_d()
          Loop While (checkContinuously=false) expression=boucle_d ≟ 1
            Set DigitalOutput pin=Cmd_Carter_Bit2; digitalValue=1
            Set DigitalOutput pin=Voyant_Table_Ga; digitalValue=0
            Set DigitalOutput pin=Voyant_Table_Dr; digitalValue=1
            Wait Sleep waitTime=0.25
            Set DigitalOutput pin=Voyant_Table_Dr; digitalValue=0
            Wait Sleep waitTime=0.25
            If SecuDroiteOk ≟  False
              Set DigitalOutput pin=Voyant_Table_Dr; digitalValue=1
              Wait Sleep waitTime=6
              If SecuDroiteOk ≟  False
                Script: close_popup()
                Wait DigitalInput pin=SecuDroiteOk; digitalValue=1
            If SecuDroiteOk ≟  True
              secu_d := 1
              Set DigitalOutput pin=Voyant_Table_Dr; digitalValue=1
              MoveJ speed 60 deg/s, acceleration 80 deg/s^2 (useActiveTCP=true) feature=Base
                Waypoint Waypoint (Variable): variable(featureName=Point_avt_initD)
                SuppressedNode
                  Waypoint Waypoint (Variable): motionParameters(blendRadius=0.006); variable(featureName=Point_init_D)
              Script: fun_execution_d()
              Set DigitalOutput pin=Cmd_Carter_Bit2; digitalValue=0
              secu_d := 0
              boucle_d := 0
          boucle := 0
        ElseIf (Pret_Table_Droi ≟ True ) and (config_d ≟ False )
          Script: close_popup()
          Popup Error (haltProgram=false message=Aucune programmation n'est actuellement detectée sur la table droite, veillez à programmer une pièce avant de vouloir l'éxécuter. inputType=Text)
          boucle := 0
SubProgram Recopie_Table_Droite (keepSynchronizedWithDisk=false)
  SuppressedNode
    URCap Path (Robotiq_Copilot, Robotiq Inc.) dataModel(NodeInitializedKey=true, urcapVersion=1.14.3, pathOptionsTypeKey=TOOL_ON_ROBOT, HackTriggeringContributionIsDefinedMethodKey=true, version=1.14.3.2973, trajectoryPath={}); state(isChildrenLocked=true)
      URCap BeforeStart Node (Robotiq_Copilot, Robotiq Inc.)
        'Insert nodes below.'
  Popup Message (haltProgram=false message=Recopie sur la table de droite  inputType=Text)
SubProgram Recopie_Table_Gauche (keepSynchronizedWithDisk=false)
  SuppressedNode
    URCap Path (Robotiq_Copilot, Robotiq Inc.) dataModel(NodeInitializedKey=true, urcapVersion=1.14.3, pathOptionsTypeKey=TOOL_ON_ROBOT, HackTriggeringContributionIsDefinedMethodKey=true, version=1.14.3.2973, trajectoryPath={}); state(isChildrenLocked=true)
      URCap BeforeStart Node (Robotiq_Copilot, Robotiq Inc.)
        'Insert nodes below.'
  Popup Message (haltProgram=false message=Recopie sur la table de gauche inputType=Text)
Thread Thread_1 (runOnlyOnce=false)
  Folder Test_Ordre_Marche [hidden by the author, left out]
  Script: sync()
Thread Thread_2 (runOnlyOnce=false)
  Folder mode_soudure [hidden by the author, left out]
  Script: sync()
Thread Thread_3 (runOnlyOnce=false)
  Folder led_cobot_2 [hidden by the author, left out]
  Script: sync()
Thread Thread_4 (runOnlyOnce=false)
  Folder led_cobot [hidden by the author, left out]
  Script: sync()
Thread Thread_5 (runOnlyOnce=false)
  Folder Test_Arc_On [hidden by the author, left out]
  Script: sync()
Thread Thread_6 (runOnlyOnce=false)
  Folder Test_Job [hidden by the author, left out]
  Script: sync()
Thread Thread_7 (runOnlyOnce=false)
  Folder secu [hidden by the author, left out]
  Script: sync()
Thread Thread_8 (runOnlyOnce=false)
  Folder bloq_soud_arret [hidden by the author, left out]
  SuppressedNode
    Folder freedrive_droit
      If led_cobot ≟  True
        If tool_in[1] ≟ True
          Script: teach_mode()
        Else 
          Script: end_teach_mode()
  Script: sync()
SuppressedNode
  Thread Thread_9 (runOnlyOnce=false)
    Folder reglage
      If reglage_d ≠0
        Script file /programs/Programmes/cobot_v2/sript/Part_reglage/REGLAGE_D.script
          |     ##############################################################################
          | 
          | ########################soudure point#########################################
          | 
          |     ##############################################################################
          | 
          |         if reglage_d == 1:                                    #remplissage tableau
          |             teach_mode()
          |             fun_popup_soud(1, 1, i)
          |             fun_front_up(adresse_bp_cobot)
          |             tab_point_app_d[i] =  get_actual_tcp_pose()     #Enregistrer position dans tableau d'approche des soudue points quand appui bouton
          |             close_popup()
          | 
          |             fun_popup_soud(2, 1, i)
          |             fun_front_up(adresse_bp_cobot)
          |             tab_point_deb_d[i] =  get_actual_tcp_pose()     #Enregistrer position debut quand appui bouton bp_cobot
          |             close_popup()
          | 
          |             tab_point_ret_d[i] = tab_point_app_d[i]         #point de retrait est le meme que le point d approche
          |             end_teach_mode()
          |             global reconfig = 1
          |             global reglage_d = 0
          | 
          |             sync()
          | 
          |         ##############################################################################
          | 
          |     ##############################################################################
          | 
          | ########################soudure lineaire######################################
          | 
          |     ##############################################################################
          | 
          |         elif reglage_d == 2:                		            #remplissage tableau
          |             teach_mode()
          |             fun_popup_soud(1, 2, j)
          |             fun_front_up(adresse_bp_cobot)
          |             tab_lin_app_d[j] =  get_actual_tcp_pose()     	#Enregistrer position dans tableau d approche des soudures lineaire quand appui Bp_cobot
          |             close_popup()
          | 
          |             fun_popup_soud(2, 2, j)
          |             fun_front_up(adresse_bp_cobot)
          |             tab_lin_deb_d[j] =  get_actual_tcp_pose()     	#Enregistrer position dans tableau debut quand appui Bp_cobot
          |             close_popup()
          | 
          |             fun_popup_soud(6, 2, j)
          |             fun_front_up(adresse_bp_cobot)
          |             tab_lin_fin_d[j] =  get_actual_tcp_pose()     	#Enregistrer position dans un tableau fin quand appui Bp_cobot
          |             close_popup()
          | 
          |             vit_lin_d[j] = fun_demande_vit(2)
          | 
          |             fun_popup_soud(7, 2, j)
          |             fun_front_up(adresse_bp_cobot)
          |             tab_lin_ret_d[j] =  get_actual_tcp_pose()     	#Enregistrer position dans tableau retrait quand appui Bp_cobot
          |             close_popup()
          |             end_teach_mode()
          |             global reglage_d = 0
          | 
          |             sync()
          | 
          |         ##############################################################################
          | 
          |     ##############################################################################
          | 
          | #########################soudure arc de cercle##################################
          | 
          |     #################################################################################
          | 
          |         elif reglage_d == 3:                                  #remplissage tableau
          |             teach_mode()
          |             fun_popup_soud(1, 3, k)
          |             fun_front_up(adresse_bp_cobot)
          |             tab_arc_app_d[k] =  get_actual_tcp_pose() 	    #Enregistrer position dans tableau d approche des soudures arc de cercle quand appui
          |             close_popup()
          | 
          |             fun_popup_soud(2, 3, k)
          |             fun_front_up(adresse_bp_cobot)
          |             tab_arc_deb_d[k] =  get_actual_tcp_pose() 	    #Enregistrer position dans tableau debut quand appui Bp_d
          |             close_popup()
          | 
          |             fun_popup_soud(4, 3, k)
          |             fun_front_up(adresse_bp_cobot)
          |             tab_arc_mil_d[k] =  get_actual_tcp_pose() 	    #Enregistrer position dans tableau milieu quand appui Bp_cobot
          |             close_popup()
          | 
          |             fun_popup_soud(6, 3, k)
          |             fun_front_up(adresse_bp_cobot)
          |             tab_arc_fin_d[k] =  get_actual_tcp_pose() 	    #Enregistrer position dans un tableau fin quand appui Bp_cobot
          |             close_popup()
          | 
          |             vit_arc_d[k] = fun_demande_vit(3)               #demande de vitesse des soudures lineaire
          | 
          |             fun_popup_soud(7, 3, k)
          |             fun_front_up(adresse_bp_cobot)
          |             tab_arc_ret_d[k] =  get_actual_tcp_pose() 	    #Enregistrer position dans tableau retrait quand appui Bp_cobot
          |             close_popup()
          |             end_teach_mode()
          |             global reglage_d = 0
          | 
          |             sync()
          | 
          |         ##############################################################################
          | 
          |     ##############################################################################
          | 
          | ############################soudure cercle####################################
          | 
          |     #################################################################################
          | 
          |         elif reglage_d == 4:                                  #remplissage tableau
          |             teach_mode()
          |             fun_popup_soud(1, 4, l)
          |             fun_front_up(adresse_bp_cobot)
          |             tab_cer_app_d[l] =  get_actual_tcp_pose()     	#Enregistrer position dans tableau d approche des soudures arc de cercle quand appui Bp_cobot
          |             close_popup()
          | 
          |             fun_popup_soud(2, 4, l)
          |             fun_front_up(adresse_bp_cobot)
          |             tab_cer_deb_d[l] =  get_actual_tcp_pose()     	#Enregistrer position dans tableau debut quand appui Bp_cobot
          |             close_popup()
          | 
          |             fun_popup_soud(3, 4, l)
          |             fun_front_up(adresse_bp_cobot)
          |             tab_cer_quart_d[l] =  get_actual_tcp_pose()   	#Enregistrer position dans tableau d'approche des soudures arc de cercle quand appui Bp_d
          |             close_popup()
          | 
          |             fun_popup_soud(4, 4, l)
          |             fun_front_up(adresse_bp_cobot)
          |             tab_cer_mil_d[l] =  get_actual_tcp_pose()     	#Enregistrer position dans tableau milieu quand appui Bp_cobot
          |             close_popup()
          | 
          |             fun_popup_soud(5, 4, l)
          |             fun_front_up(adresse_bp_cobot)
          |             tab_cer_tro_d[l] =  get_actual_tcp_pose()     	#Enregistrer position dans tableau milieu quand appui Bp_cobot
          |             close_popup()
          | 
          |             fun_popup_soud(6, 4, l)
          |             fun_front_up(adresse_bp_cobot)
          |             tab_cer_fin_d[l] =  get_actual_tcp_pose()     	#Enregistrer position dans un tableau fin quand appui Bp_cobot
          |             close_popup()
          | 
          |             vit_cer_d[l] = fun_demande_vit(4)
          | 
          |             fun_popup_soud(7, 4, l)
          |             fun_front_up(adresse_bp_cobot)
          |             tab_cer_ret_d[l] =  get_actual_tcp_pose()    	#position de retrait est la meme que position d approche
          |             close_popup()
          |             end_teach_mode()
          |             global reglage_d = 0
          |             sync()
          | 
          |         end
          | 
          |     ##############################################################################
          | 
          | ############################################################
        Script: sync()
      If reglage_g ≠0
        Script file /programs/usbdisk_0/COBOT/finish/reg/REGLAGE_G.script
          |     ##############################################################################
          | 
          | ########################soudure point#########################################
          | 
          |     ##############################################################################
          | 
          |         if reglage_g == 1:                                    #remplissage tableau
          |             teach_mode()
          |             fun_popup_soud(1, 1, i)
          |             fun_front_up(adresse_bp_cobot)
          |             tab_point_app_g[i] =  get_actual_tcp_pose()     #Enregistrer position dans tableau d'approche des soudue points quand appui bouton
          |             close_popup()
          | 
          |             fun_popup_soud(2, 1, i)
          |             fun_front_up(adresse_bp_cobot)
          |             tab_point_deb_g[i] =  get_actual_tcp_pose()     #Enregistrer position debut quand appui bouton bp_cobot
          |             close_popup()
          | 
          |             tab_point_ret_g[i] = tab_point_app_g[i]         #point de retrait est le meme que le point d approche
          |             end_teach_mode()
          |             global reconfig = 1
          |             global reglage_g = 0
          | 
          |             sync()
          | 
          |         ##############################################################################
          | 
          |     ##############################################################################
          | 
          | ########################soudure lineaire######################################
          | 
          |     ##############################################################################
          | 
          |         elif reglage_g == 2:                		            #remplissage tableau
          |             teach_mode()
          |             fun_popup_soud(1, 2, j)
          |             fun_front_up(adresse_bp_cobot)
          |             tab_lin_app_g[j] =  get_actual_tcp_pose()     	#Enregistrer position dans tableau d approche des soudures lineaire quand appui Bp_cobot
          |             close_popup()
          | 
          |             fun_popup_soud(2, 2, j)
          |             fun_front_up(adresse_bp_cobot)
          |             tab_lin_deb_g[j] =  get_actual_tcp_pose()     	#Enregistrer position dans tableau debut quand appui Bp_cobot
          |             close_popup()
          | 
          |             fun_popup_soud(6, 2, j)
          |             fun_front_up(adresse_bp_cobot)
          |             tab_lin_fin_g[j] =  get_actual_tcp_pose()     	#Enregistrer position dans un tableau fin quand appui Bp_cobot
          |             close_popup()
          | 
          |             vit_lin_g[j] = fun_demande_vit(2)
          | 
          |             fun_popup_soud(7, 2, j)
          |             fun_front_up(adresse_bp_cobot)
          |             tab_lin_ret_g[j] =  get_actual_tcp_pose()     	#Enregistrer position dans tableau retrait quand appui Bp_cobot
          |             close_popup()
          |             end_teach_mode()
          |             global reglage_g = 0
          | 
          |             sync()
          | 
          |         ##############################################################################
          | 
          |     ##############################################################################
          | 
          | #########################soudure arc de cercle##################################
          | 
          |     #################################################################################
          | 
          |         elif reglage_g == 3:                                  #remplissage tableau
          |             teach_mode()
          |             fun_popup_soud(1, 3, k)
          |             fun_front_up(adresse_bp_cobot)
          |             tab_arc_app_g[k] =  get_actual_tcp_pose() 	    #Enregistrer position dans tableau d approche des soudures arc de cercle quand appui
          |             close_popup()
          | 
          |             fun_popup_soud(2, 3, k)
          |             fun_front_up(adresse_bp_cobot)
          |             tab_arc_deb_g[k] =  get_actual_tcp_pose() 	    #Enregistrer position dans tableau debut quand appui BP_cobot
          |             close_popup()
          | 
          |             fun_popup_soud(4, 3, k)
          |             fun_front_up(adresse_bp_cobot)
          |             tab_arc_mil_g[k] =  get_actual_tcp_pose() 	    #Enregistrer position dans tableau milieu quand appui Bp_cobot
          |             close_popup()
          | 
          |             fun_popup_soud(6, 3, k)
          |             fun_front_up(adresse_bp_cobot)
          |             tab_arc_fin_g[k] =  get_actual_tcp_pose() 	    #Enregistrer position dans un tableau fin quand appui Bp_cobot
          |             close_popup()
          | 
          |             vit_arc_g[k] = fun_demande_vit(3)               #demande de vitesse des soudures lineaire
          | 
          |             fun_popup_soud(7, 3, k)
          |             fun_front_up(adresse_bp_cobot)
          |             tab_arc_ret_g[k] =  get_actual_tcp_pose() 	    #Enregistrer position dans tableau retrait quand appui Bp_cobot
          |             close_popup()
          |             end_teach_mode()
          |             global reglage_g = 0
          | 
          |             sync()
          | 
          |         ##############################################################################
          | 
          |     ##############################################################################
          | 
          | ############################soudure cercle####################################
          | 
          |     #################################################################################
          | 
          |         elif reglage_g == 4:                                  #remplissage tableau
          |             teach_mode()
          |             fun_popup_soud(1, 4, l)
          |             fun_front_up(adresse_bp_cobot)
          |             tab_cer_app_g[l] =  get_actual_tcp_pose()     	#Enregistrer position dans tableau d approche des soudures arc de cercle quand appui Bp_cobot
          |             close_popup()
          | 
          |             fun_popup_soud(2, 4, l)
          |             fun_front_up(adresse_bp_cobot)
          |             tab_cer_deb_g[l] =  get_actual_tcp_pose()     	#Enregistrer position dans tableau debut quand appui Bp_cobot
          |             close_popup()
          | 
          |             fun_popup_soud(3, 4, l)
          |             fun_front_up(adresse_bp_cobot)
          |             tab_cer_quart_g[l] =  get_actual_tcp_pose()   	#Enregistrer position dans tableau d'approche des soudures arc de cercle quand appui Bp_cobot
          |             close_popup()
          | 
          |             fun_popup_soud(4, 4, l)
          |             fun_front_up(adresse_bp_cobot)
          |             tab_cer_mil_g[l] =  get_actual_tcp_pose()     	#Enregistrer position dans tableau milieu quand appui Bp_cobot
          |             close_popup()
          | 
          |             fun_popup_soud(5, 4, l)
          |             fun_front_up(adresse_bp_cobot)
          |             tab_cer_tro_g[l] =  get_actual_tcp_pose()     	#Enregistrer position dans tableau milieu quand appui Bp_cobot
          |             close_popup()
          | 
          |             fun_popup_soud(6, 4, l)
          |             fun_front_up(adresse_bp_cobot)
          |             tab_cer_fin_g[l] =  get_actual_tcp_pose()     	#Enregistrer position dans un tableau fin quand appui Bp_cobot
          |             close_popup()
          | 
          |             vit_cer_g[l] = fun_demande_vit(4)
          | 
          |             fun_popup_soud(7, 4, l)
          |             fun_front_up(adresse_bp_cobot)
          |             tab_cer_ret_g[l] =  get_actual_tcp_pose()    	#position de retrait est la meme que position d approche
          |             close_popup()
          |             end_teach_mode()
          |             global reglage_g = 0
          |             sync()
          | 
          |         end
          | 
          |     ##############################################################################
          | 
          | ############################################################
        Script: sync()
      Script: sync()
    Script: sync()
Thread Thread_10 (runOnlyOnce=false)
  Folder reglage [hidden by the author, left out]
  Script: sync()
